FUNCTION_BLOCK FB_ProtoWriter
VAR_INPUT
END_VAR
VAR_OUTPUT
END_VAR
VAR
	_pBuffer    	: POINTER TO BYTE;
	_nCapacity  	: UDINT;
	_nLength    	: UDINT;
	_bError     	: BOOL;
END_VAR

// Pointer to the start of the encoded bytes. Valid until the next Init call.
PROPERTY Buffer : POINTER TO BYTE
GET
Buffer := _pBuffer;
END_GET
END_PROPERTY

PROPERTY HasError : BOOL
GET
HasError := _bError;
END_GET
END_PROPERTY

METHOD Init
VAR_INPUT
	pBuffer		 		: POINTER TO BYTE;
	nCapacity			: UDINT;
END_VAR
_pBuffer   := pBuffer;
_nCapacity := nCapacity;
_nLength   := 0;
_bError    := FALSE;
END_METHOD

PROPERTY Length : UDINT
GET
Length := _nLength;
END_GET
END_PROPERTY

METHOD Reset : PVOID
VAR_INPUT
END_VAR
_nLength := 0;
_bError  := FALSE;
END_METHOD

METHOD PUBLIC WriteBool : BOOL
VAR_INPUT
	nFieldNumber 	: UDINT;
	bValue       	: BOOL;
END_VAR
WriteBool := writeTag(nFieldNumber, E_ProtoWireType.Varint)
	AND writeVarint(BOOL_TO_ULINT(bValue));
END_METHOD

METHOD PUBLIC WriteBytes : BOOL
VAR_INPUT
	nFieldNumber 	: UDINT;
	pData        	: POINTER TO BYTE;
	nLen         	: UDINT;
END_VAR
WriteBytes := writeTag(nFieldNumber, E_ProtoWireType.LengthDelimited)
	AND writeVarint(UDINT_TO_ULINT(nLen))
	AND writeRawBytes(pData, nLen);
END_METHOD

METHOD PUBLIC WriteDouble : BOOL
VAR_INPUT
	nFieldNumber 	: UDINT;
	fValue       	: LREAL;
END_VAR
VAR
	nRaw			: LWORD;
END_VAR
MEMCPY(destAddr := ADR(nRaw), srcAddr := ADR(fValue), n := 8);
WriteDouble := writeTag(nFieldNumber, E_ProtoWireType.Fixed64)
	AND writeRawBytes(ADR(nRaw), 8);
END_METHOD

METHOD PUBLIC WriteFloat : BOOL
VAR_INPUT
	nFieldNumber 	: UDINT;
	fValue       	: REAL;
END_VAR
VAR
	nRaw			: DWORD;
END_VAR
MEMCPY(destAddr := ADR(nRaw), srcAddr := ADR(fValue), n := 4);
WriteFloat := writeTag(nFieldNumber, E_ProtoWireType.Fixed32)
	AND writeRawBytes(ADR(nRaw), 4);
END_METHOD

METHOD PRIVATE writeRawByte : BOOL
VAR_INPUT
	nByte		: BYTE;
END_VAR
IF _bError OR _nLength >= _nCapacity THEN
	_bError := TRUE;
	writeRawByte := FALSE;
	RETURN;
END_IF
_pBuffer[_nLength] := nByte;
_nLength := _nLength + 1;
writeRawByte := TRUE;
END_METHOD

METHOD PRIVATE writeRawBytes : BOOL
VAR_INPUT
	pData : POINTER TO BYTE;
	nLen  : UDINT;
END_VAR
IF _bError OR (_nLength + nLen > _nCapacity) THEN
	_bError := TRUE;
	writeRawBytes := FALSE;
	RETURN;
END_IF
MEMCPY(destAddr := _pBuffer + _nLength, srcAddr := pData, n := nLen);
_nLength := _nLength + nLen;
writeRawBytes := TRUE;
END_METHOD

METHOD PUBLIC WriteString : BOOL
VAR_INPUT
	nFieldNumber 	: UDINT;
	sValue       	: STRING(255);
END_VAR
VAR
	nLen			: INT;
END_VAR
nLen := LEN(sValue);
WriteString := writeTag(nFieldNumber, E_ProtoWireType.LengthDelimited)
	AND writeVarint(TO_ULINT(nLen))
	AND writeRawBytes(ADR(sValue), TO_UDINT(nLen));
END_METHOD

METHOD PRIVATE writeTag : BOOL
VAR_INPUT
	nFieldNumber 	: UDINT;
	eWireType    	: E_ProtoWireType;
END_VAR
writeTag := writeVarint(
	SHL(UDINT_TO_ULINT(nFieldNumber), 3) OR INT_TO_ULINT(TO_INT(eWireType))
);
END_METHOD

METHOD PUBLIC WriteUInt32 : BOOL
VAR_INPUT
	nFieldNumber 	: UDINT;
	nValue       	: UDINT;
END_VAR
WriteUInt32 := writeTag(nFieldNumber, E_ProtoWireType.Varint)
	AND writeVarint(UDINT_TO_ULINT(nValue));
END_METHOD

METHOD PUBLIC WriteUInt64 : BOOL
VAR_INPUT
	nFieldNumber 	: UDINT;
  	nValue       	: ULINT;
END_VAR
WriteUInt64 := writeTag(nFieldNumber, E_ProtoWireType.Varint)
	AND writeVarint(nValue);
END_METHOD

METHOD PRIVATE writeVarint : BOOL
VAR_INPUT
	nValue		: ULINT;
END_VAR
VAR
	nByte		: BYTE;
END_VAR
IF _bError THEN writeVarint := FALSE; RETURN; END_IF
REPEAT
	nByte  := ULINT_TO_BYTE(nValue AND 16#7F);
	nValue := SHR(nValue, 7);
	IF nValue <> 0 THEN
  		nByte := nByte OR 16#80;  // more bytes follow
	END_IF
	IF NOT writeRawByte(nByte) THEN
		writeVarint := FALSE;
		RETURN;
	END_IF
UNTIL nValue = 0
END_REPEAT;
writeVarint := TRUE;
END_METHOD

END_FUNCTION_BLOCK

(* stored: Version 1.1.0.1
   POU FB_ProtoWriter: Id {04ab8747-175c-4210-9303-f7a14ac341c4}, SpecialFunc None
   Property Buffer: Id {a1a1a1a1-b2b2-c3c3-d4d4-e5e5e5e5e5e5}
   Get Get: Id {f6f6f6f6-a7a7-b8b8-c9c9-d0d0d0d0d0d0}
   Property HasError: Id {314238dd-6eee-42f6-bdcf-e3c3aadea4f9}
   Get Get: Id {fcb31419-c09b-4143-aabb-c2d73b254ea8}
   Method Init: Id {7b9e04db-136b-4dda-929d-c27fc11952fe}
   Property Length: Id {f04fe5aa-6644-4156-8899-2e8eca6bf4cc}
   Get Get: Id {522ced7a-ffe5-4ee5-bfa5-717a98316592}
   Method Reset: Id {dcb2ef2c-08c0-4846-859a-6d23915ac1b7}
   Method WriteBool: Id {156c21b2-30c8-413b-bdb2-84f74a1f38e0}
   Method WriteBytes: Id {f6d80a59-5b99-4b8c-8754-675d4e12b293}
   Method WriteDouble: Id {bfeefe92-e14e-42d5-b70a-866f3d07ab09}
   Method WriteFloat: Id {928610a2-c597-44dc-bb0c-5db4bf56c895}
   Method writeRawByte: Id {96d19778-a498-4581-89e6-cd2fe0547295}
   Method writeRawBytes: Id {d5ba1cdf-dccf-4324-b6a9-0bc2bb6c677f}
   Method WriteString: Id {fc92f74d-e092-4e01-8280-ac8903069ea2}
   Method writeTag: Id {11904569-014c-438a-b1c0-95da59f70072}
   Method WriteUInt32: Id {faf32b82-ad32-4dce-b276-2d0533a72c9e}
   Method WriteUInt64: Id {557877d0-3fc8-474c-908e-9f5131acbe2a}
   Method writeVarint: Id {a78d27d9-7258-4763-ae70-8b4ec8dd8ca3} *)
